ABB RAPID module: Module1.mod

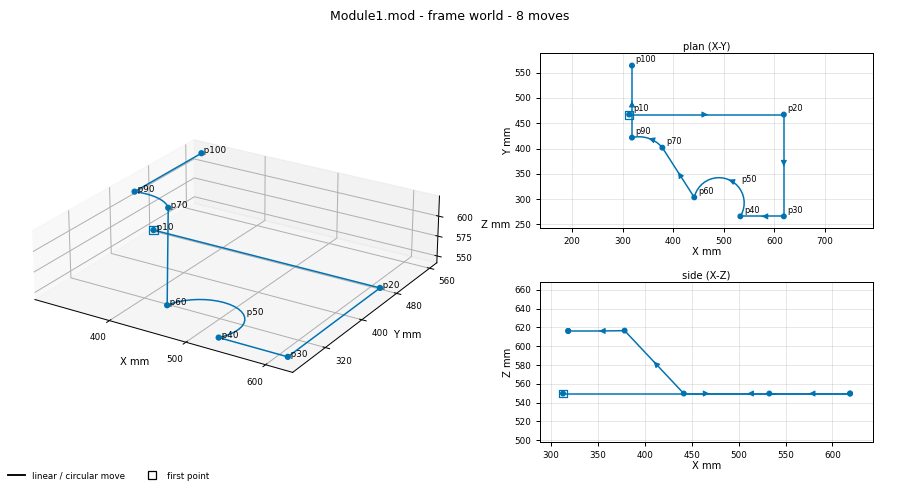
[picture p0: tool path of Module1.mod in frame world, 8 of 10 moves have a stored position in this frame; points joined in program order, loops and branches not executed]
MODULE Module1
	CONST jointtarget jpos10:=[[65.3885,-46.5801,47.724,180.577,-28.1733,-181.532],[9E+9,9E+9,9E+9,9E+9,9E+9,9E+9]];
	CONST robtarget p10:=[[312.95,467.14,549.66],[0.426451,-0.473639,0.72144,0.270795],[0,3,-4,1],[9E+9,9E+9,9E+9,9E+9,9E+9,9E+9]];
	CONST robtarget p20:=[[618.74,467.14,549.66],[0.42645,-0.473638,0.721441,0.270796],[0,3,-4,1],[9E+9,9E+9,9E+9,9E+9,9E+9,9E+9]];
	CONST robtarget p30:=[[618.74,265.86,549.66],[0.42645,-0.473638,0.721441,0.270796],[0,3,-4,1],[9E+9,9E+9,9E+9,9E+9,9E+9,9E+9]];
	CONST robtarget p40:=[[532.78,265.86,549.66],[0.42645,-0.473638,0.721441,0.270796],[0,3,-4,1],[9E+9,9E+9,9E+9,9E+9,9E+9,9E+9]];
	CONST robtarget p60:=[[441.64,303.39,549.66],[0.42645,-0.473639,0.721441,0.270795],[0,3,-4,1],[9E+9,9E+9,9E+9,9E+9,9E+9,9E+9]];
	CONST robtarget p50:=[[527.00,326.42,549.66],[0.42645,-0.473638,0.721441,0.270795],[0,3,-4,1],[9E+9,9E+9,9E+9,9E+9,9E+9,9E+9]];
	CONST robtarget p70:=[[378.59,401.65,616.69],[0.282515,-0.571295,0.767786,0.0656612],[0,2,-3,1],[9E+9,9E+9,9E+9,9E+9,9E+9,9E+9]];
	CONST robtarget p90:=[[318.51,421.57,616.31],[0.282515,-0.571296,0.767786,0.0656604],[0,1,-3,1],[9E+9,9E+9,9E+9,9E+9,9E+9,9E+9]];
	CONST robtarget p80:=[[352.21,419.85,616.31],[0.282515,-0.571296,0.767786,0.0656606],[0,1,-3,1],[9E+9,9E+9,9E+9,9E+9,9E+9,9E+9]];
	CONST robtarget p100:=[[318.51,564.09,616.31],[0.282515,-0.571296,0.767786,0.0656605],[0,1,-2,1],[9E+9,9E+9,9E+9,9E+9,9E+9,9E+9]];
	CONST jointtarget jpos20:=[[61.3922,-19.5959,59.1382,159.2,-18.4118,-174.012],[9E+9,9E+9,9E+9,9E+9,9E+9,9E+9]];
    !***********************************************************
    !
    ! Module:  Module1
    !
    ! Description:
    !   <Insert description here>
    !
    ! Author: cyx
    !
    ! Version: 1.0
    !
    !***********************************************************


    !***********************************************************
    !
    ! Procedure main
    !
    !   This is the entry point of your program
    !
    !***********************************************************
    PROC main()
        MoveAbsJ jpos10\NoEOffs, v1000, z50, tool0;
        !Add your code here
        MoveJ p10, v1000, fine, tool0;
        MoveL p20, v1000, fine, tool0;
        MoveL p30, v1000, fine, tool0;
        MoveL p40, v1000, fine, tool0;
        MoveC p50, p60, v1000, fine, tool0;
        MoveL p70, v1000, fine, tool0;
        MoveC p80, p90, v1000, fine, tool0;
        MoveL p100, v1000, fine, tool0;
        MoveAbsJ jpos10\NoEOffs, v1000, fine, tool0;
    ENDPROC
ENDMODULE
